FUNCTION_BLOCK FB_Blink
VAR_INPUT
	bEnable : BOOL; // Startsignal für Blinken
	PT : TIME; // Periodendauer des Blinklichts
END_VAR
VAR_OUTPUT
	bBlink : BOOL := FALSE; // Blinksignal
END_VAR
VAR
	fbTon : TON; // einschaltverzögerung
	fbTP : TP; // Pulsetimer
END_VAR

// FUnktionsbaustein ausführen
fbTon(IN:= , PT:= , Q=> , ET=> );
fbTP(IN:= , PT:= , Q=> , ET=> );

// zyklisches ausführen von TON
fbTon.IN := bEnable AND NOT fbTon.Q;
fbTon.PT := PT;

// Pulsen von bBlink nach TON.Q = True
fbTP.IN := fbTon.Q; // Ausgang von fbTon.Q triggert den fbTP.IN
fbTP.PT := PT/2;
bBlink := fbTP.Q;

END_FUNCTION_BLOCK

(* stored: Version 1.1.0.1
   POU FB_Blink: Id {a5e903be-f4ae-4f09-bf7b-8da8294f9ea2}, SpecialFunc None *)
